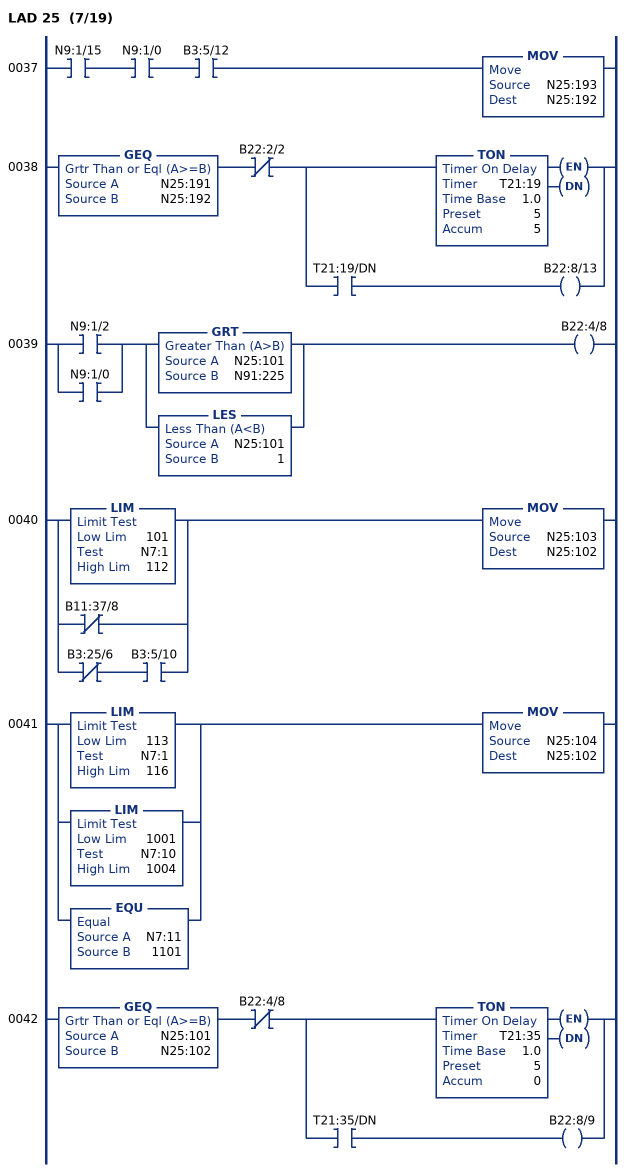
% Rung: 37 %
SOR XIC N9:1/15 XIC N9:1/0 XIC B3:5/12 MOV N25:193 N25:192 EOR
% Rung: 38 %
SOR GEQ N25:191 N25:192 XIO B22:2/2 BST TON T21:19 1.0 5 5 NXB XIC T21:19/DN OTE B22:8/13 BND EOR
% Rung: 39 %
SOR BST XIC N9:1/2 NXB XIC N9:1/0 BND BST GRT N25:101 N91:225 NXB LES N25:101 1 BND OTE B22:4/8 EOR
% Rung: 40 %
SOR BST LIM 101 N7:1 112 NXB XIO B11:37/8 NXB XIO B3:25/6 XIC B3:5/10 BND MOV N25:103 N25:102 EOR
% Rung: 41 %
SOR BST LIM 113 N7:1 116 NXB LIM 1001 N7:10 1004 NXB EQU N7:11 1101 BND MOV N25:104 N25:102 EOR
% Rung: 42 %
SOR GEQ N25:101 N25:102 XIO B22:4/8 BST TON T21:35 1.0 5 0 NXB XIC T21:35/DN OTE B22:8/9 BND EOR

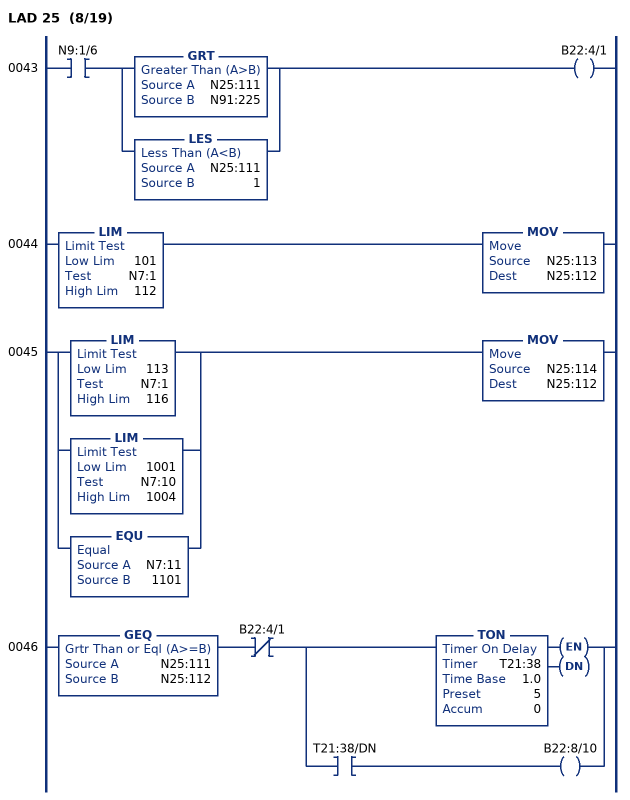
% Rung: 43 %
SOR XIC N9:1/6 BST GRT N25:111 N91:225 NXB LES N25:111 1 BND OTE B22:4/1 EOR
% Rung: 44 %
SOR LIM 101 N7:1 112 MOV N25:113 N25:112 EOR
% Rung: 45 %
SOR BST LIM 113 N7:1 116 NXB LIM 1001 N7:10 1004 NXB EQU N7:11 1101 BND MOV N25:114 N25:112 EOR
% Rung: 46 %
SOR GEQ N25:111 N25:112 XIO B22:4/1 BST TON T21:38 1.0 5 0 NXB XIC T21:38/DN OTE B22:8/10 BND EOR

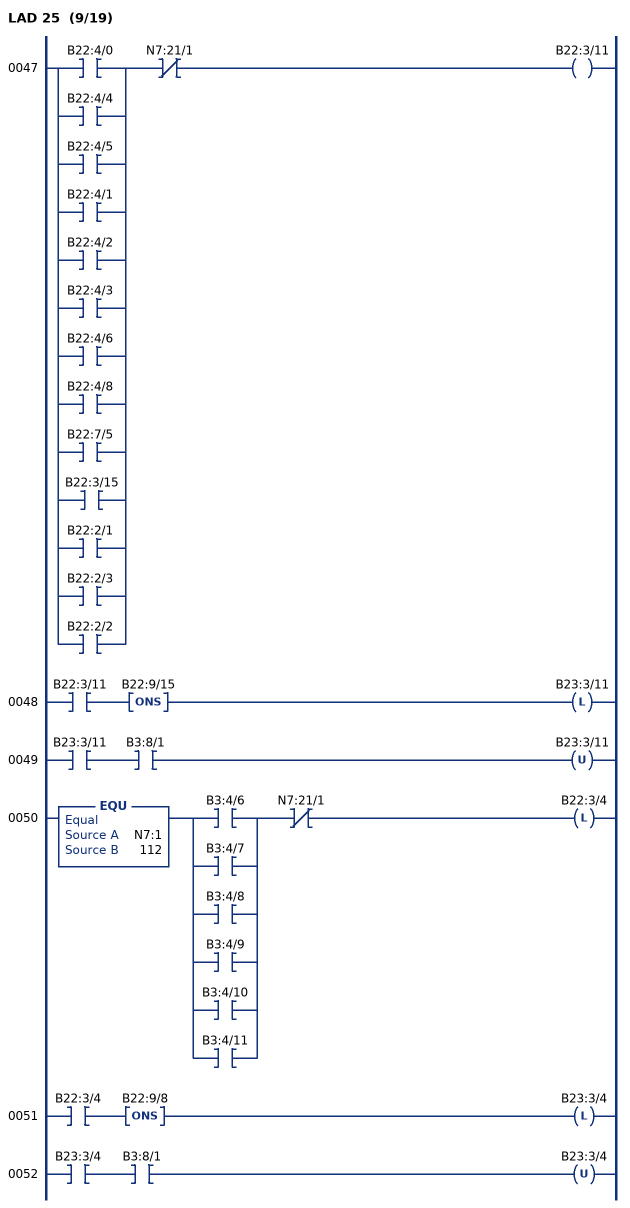
% Rung: 47 %
SOR BST XIC B22:4/0 NXB XIC B22:4/4 NXB XIC B22:4/5 NXB XIC B22:4/1 NXB XIC B22:4/2 NXB XIC B22:4/3 NXB XIC B22:4/6 NXB XIC B22:4/8 NXB XIC B22:7/5 NXB XIC B22:3/15 NXB XIC B22:2/1 NXB XIC B22:2/3 NXB XIC B22:2/2 BND XIO N7:21/1 OTE B22:3/11 EOR
% Rung: 48 %
SOR XIC B22:3/11 OSR B22:9/15 OTL B23:3/11 EOR
% Rung: 49 %
SOR XIC B23:3/11 XIC B3:8/1 OTU B23:3/11 EOR
% Rung: 50 %
SOR EQU N7:1 112 BST XIC B3:4/6 NXB XIC B3:4/7 NXB XIC B3:4/8 NXB XIC B3:4/9 NXB XIC B3:4/10 NXB XIC B3:4/11 BND XIO N7:21/1 OTL B22:3/4 EOR
% Rung: 51 %
SOR XIC B22:3/4 OSR B22:9/8 OTL B23:3/4 EOR
% Rung: 52 %
SOR XIC B23:3/4 XIC B3:8/1 OTU B23:3/4 EOR

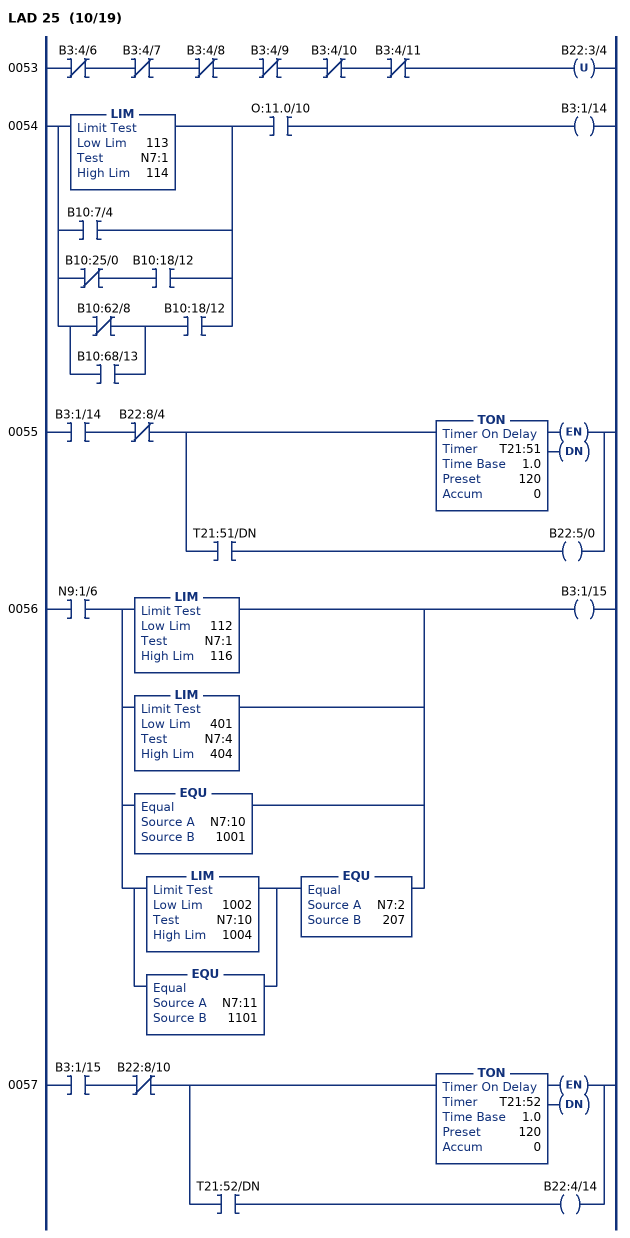
% Rung: 53 %
SOR XIO B3:4/6 XIO B3:4/7 XIO B3:4/8 XIO B3:4/9 XIO B3:4/10 XIO B3:4/11 OTU B22:3/4 EOR
% Rung: 54 %
SOR BST LIM 113 N7:1 114 NXB XIC B10:7/4 NXB XIO B10:25/0 XIC B10:18/12 NXB BST XIO B10:62/8 NXB XIC B10:68/13 BND XIC B10:18/12 BND XIC O:11.0/10 OTE B3:1/14 EOR
% Rung: 55 %
SOR XIC B3:1/14 XIO B22:8/4 BST TON T21:51 1.0 120 0 NXB XIC T21:51/DN OTE B22:5/0 BND EOR
% Rung: 56 %
SOR XIC N9:1/6 BST LIM 112 N7:1 116 NXB LIM 401 N7:4 404 NXB EQU N7:10 1001 NXB BST LIM 1002 N7:10 1004 NXB EQU N7:11 1101 BND EQU N7:2 207 BND OTE B3:1/15 EOR
% Rung: 57 %
SOR XIC B3:1/15 XIO B22:8/10 BST TON T21:52 1.0 120 0 NXB XIC T21:52/DN OTE B22:4/14 BND EOR

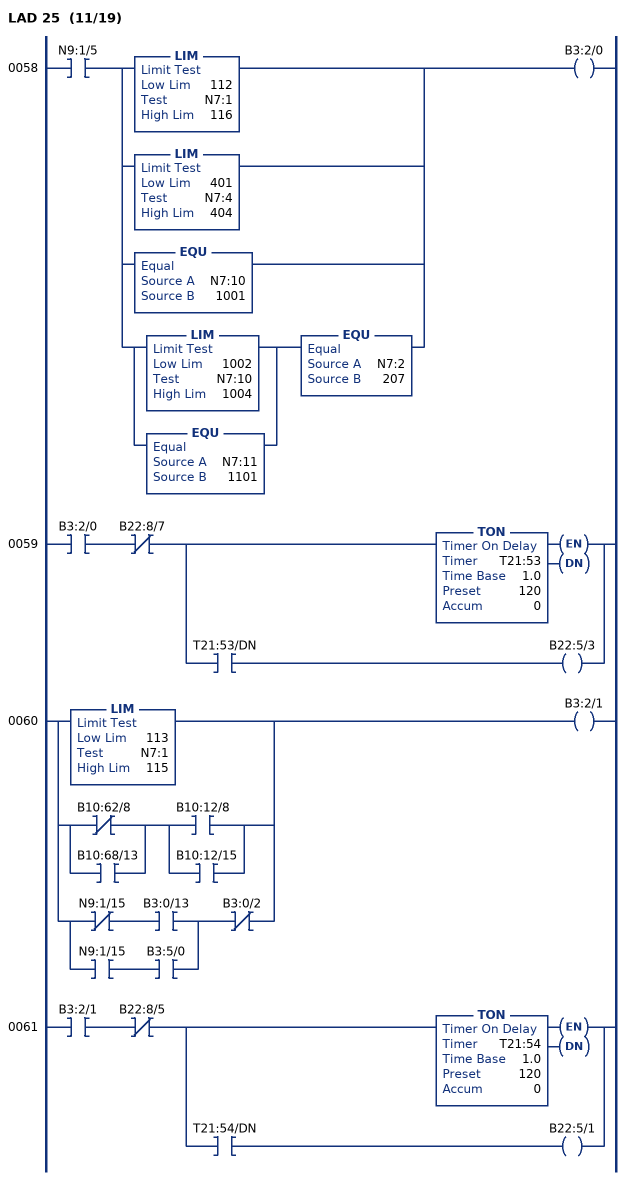
% Rung: 58 %
SOR XIC N9:1/5 BST LIM 112 N7:1 116 NXB LIM 401 N7:4 404 NXB EQU N7:10 1001 NXB BST LIM 1002 N7:10 1004 NXB EQU N7:11 1101 BND EQU N7:2 207 BND OTE B3:2/0 EOR
% Rung: 59 %
SOR XIC B3:2/0 XIO B22:8/7 BST TON T21:53 1.0 120 0 NXB XIC T21:53/DN OTE B22:5/3 BND EOR
% Rung: 60 %
SOR BST LIM 113 N7:1 115 NXB BST XIO B10:62/8 NXB XIC B10:68/13 BND BST XIC B10:12/8 NXB XIC B10:12/15 BND NXB BST XIO N9:1/15 XIC B3:0/13 NXB XIC N9:1/15 XIC B3:5/0 BND XIO B3:0/2 BND OTE B3:2/1 EOR
% Rung: 61 %
SOR XIC B3:2/1 XIO B22:8/5 BST TON T21:54 1.0 120 0 NXB XIC T21:54/DN OTE B22:5/1 BND EOR

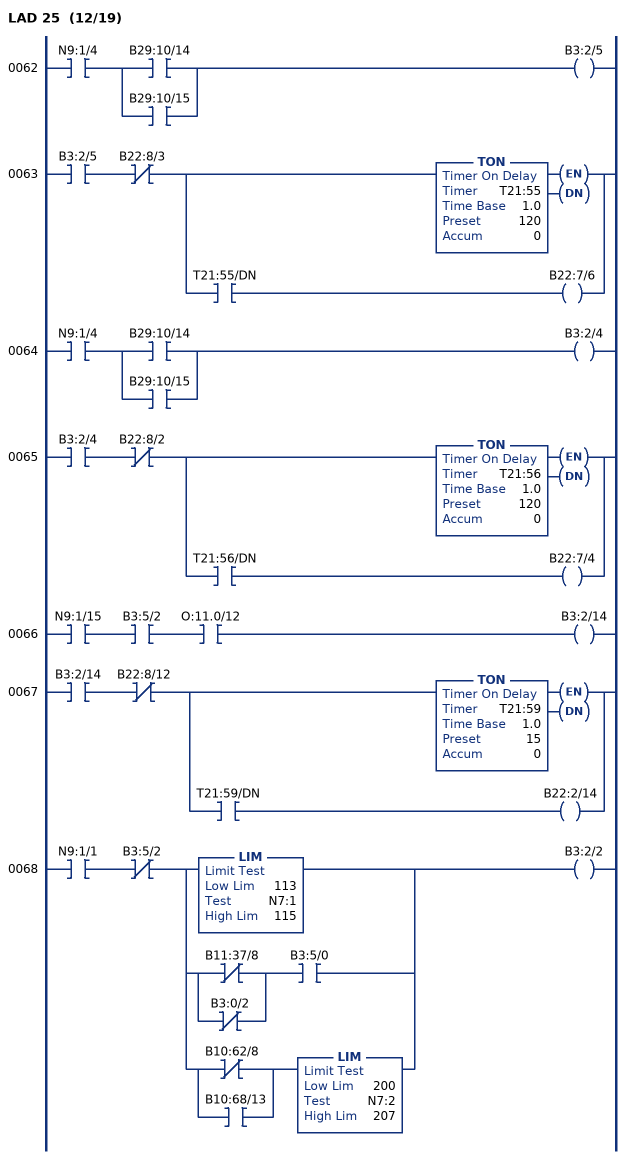
% Rung: 62 %
SOR XIC N9:1/4 BST XIC B29:10/14 NXB XIC B29:10/15 BND OTE B3:2/5 EOR
% Rung: 63 %
SOR XIC B3:2/5 XIO B22:8/3 BST TON T21:55 1.0 120 0 NXB XIC T21:55/DN OTE B22:7/6 BND EOR
% Rung: 64 %
SOR XIC N9:1/4 BST XIC B29:10/14 NXB XIC B29:10/15 BND OTE B3:2/4 EOR
% Rung: 65 %
SOR XIC B3:2/4 XIO B22:8/2 BST TON T21:56 1.0 120 0 NXB XIC T21:56/DN OTE B22:7/4 BND EOR
% Rung: 66 %
SOR XIC N9:1/15 XIC B3:5/2 XIC O:11.0/12 OTE B3:2/14 EOR
% Rung: 67 %
SOR XIC B3:2/14 XIO B22:8/12 BST TON T21:59 1.0 15 0 NXB XIC T21:59/DN OTE B22:2/14 BND EOR
% Rung: 68 %
SOR XIC N9:1/1 XIO B3:5/2 BST LIM 113 N7:1 115 NXB BST XIO B11:37/8 NXB XIO B3:0/2 BND XIC B3:5/0 NXB BST XIO B10:62/8 NXB XIC B10:68/13 BND LIM 200 N7:2 207 BND OTE B3:2/2 EOR

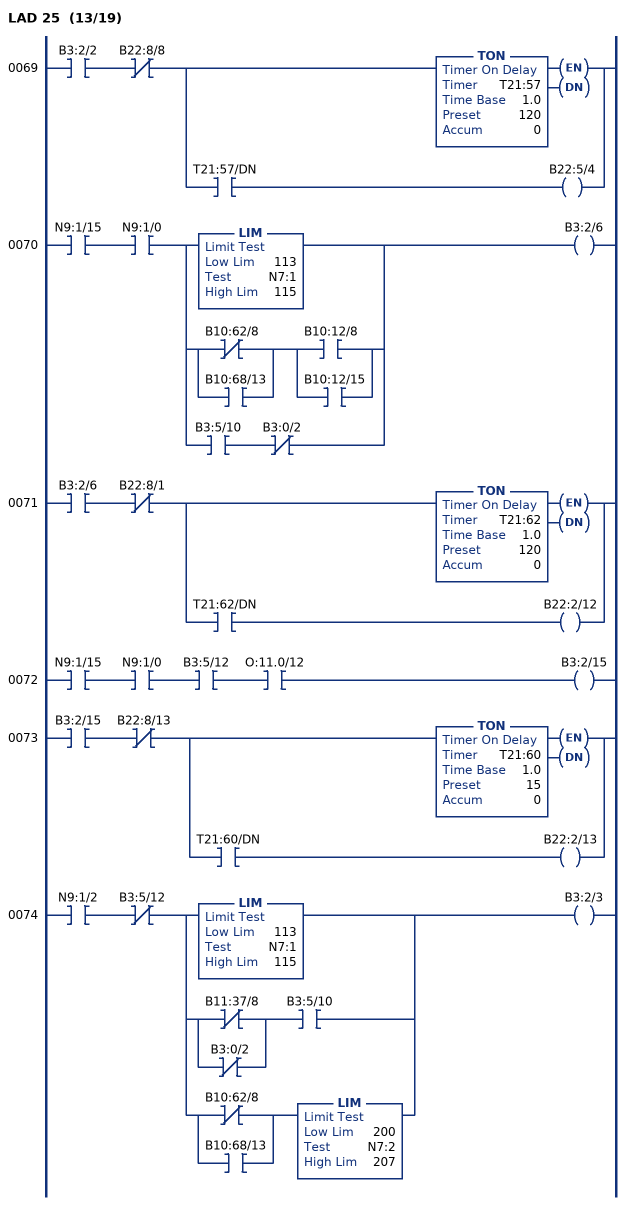
% Rung: 69 %
SOR XIC B3:2/2 XIO B22:8/8 BST TON T21:57 1.0 120 0 NXB XIC T21:57/DN OTE B22:5/4 BND EOR
% Rung: 70 %
SOR XIC N9:1/15 XIC N9:1/0 BST LIM 113 N7:1 115 NXB BST XIO B10:62/8 NXB XIC B10:68/13 BND BST XIC B10:12/8 NXB XIC B10:12/15 BND NXB XIC B3:5/10 XIO B3:0/2 BND OTE B3:2/6 EOR
% Rung: 71 %
SOR XIC B3:2/6 XIO B22:8/1 BST TON T21:62 1.0 120 0 NXB XIC T21:62/DN OTE B22:2/12 BND EOR
% Rung: 72 %
SOR XIC N9:1/15 XIC N9:1/0 XIC B3:5/12 XIC O:11.0/12 OTE B3:2/15 EOR
% Rung: 73 %
SOR XIC B3:2/15 XIO B22:8/13 BST TON T21:60 1.0 15 0 NXB XIC T21:60/DN OTE B22:2/13 BND EOR
% Rung: 74 %
SOR XIC N9:1/2 XIO B3:5/12 BST LIM 113 N7:1 115 NXB BST XIO B11:37/8 NXB XIO B3:0/2 BND XIC B3:5/10 NXB BST XIO B10:62/8 NXB XIC B10:68/13 BND LIM 200 N7:2 207 BND OTE B3:2/3 EOR

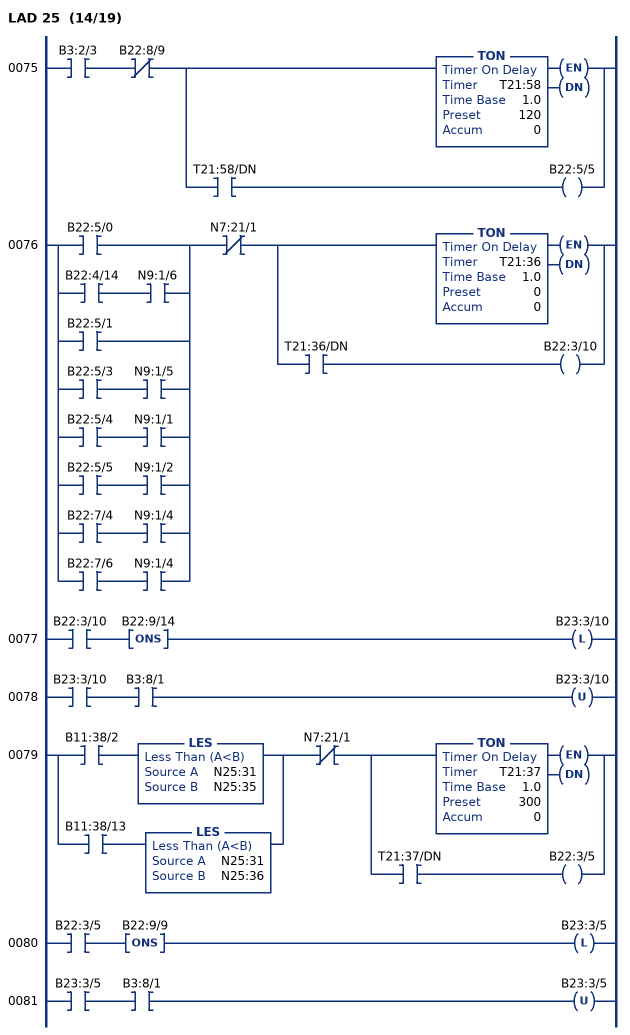
% Rung: 75 %
SOR XIC B3:2/3 XIO B22:8/9 BST TON T21:58 1.0 120 0 NXB XIC T21:58/DN OTE B22:5/5 BND EOR
% Rung: 76 %
SOR BST XIC B22:5/0 NXB XIC B22:4/14 XIC N9:1/6 NXB XIC B22:5/1 NXB XIC B22:5/3 XIC N9:1/5 NXB XIC B22:5/4 XIC N9:1/1 NXB XIC B22:5/5 XIC N9:1/2 NXB XIC B22:7/4 XIC N9:1/4 NXB XIC B22:7/6 XIC N9:1/4 BND XIO N7:21/1 BST TON T21:36 1.0 0 0 NXB XIC T21:36/DN OTE B22:3/10 BND EOR
% Rung: 77 %
SOR XIC B22:3/10 OSR B22:9/14 OTL B23:3/10 EOR
% Rung: 78 %
SOR XIC B23:3/10 XIC B3:8/1 OTU B23:3/10 EOR
% Rung: 79 %
SOR BST XIC B11:38/2 LES N25:31 N25:35 NXB XIC B11:38/13 LES N25:31 N25:36 BND XIO N7:21/1 BST TON T21:37 1.0 300 0 NXB XIC T21:37/DN OTE B22:3/5 BND EOR
% Rung: 80 %
SOR XIC B22:3/5 OSR B22:9/9 OTL B23:3/5 EOR
% Rung: 81 %
SOR XIC B23:3/5 XIC B3:8/1 OTU B23:3/5 EOR

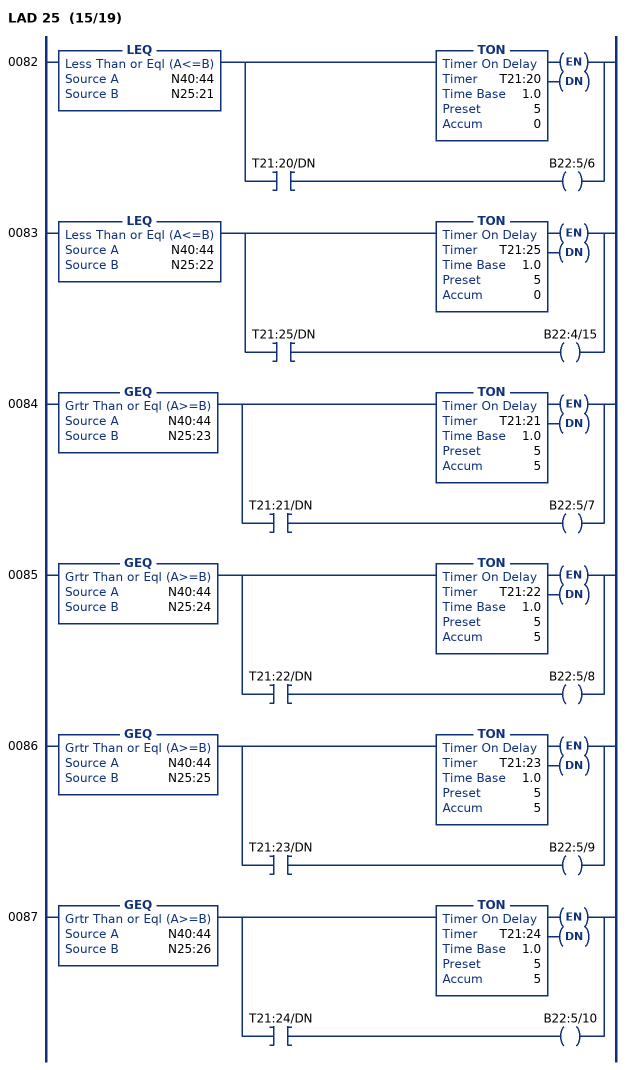
% Rung: 82 %
SOR LEQ N40:44 N25:21 BST TON T21:20 1.0 5 0 NXB XIC T21:20/DN OTE B22:5/6 BND EOR
% Rung: 83 %
SOR LEQ N40:44 N25:22 BST TON T21:25 1.0 5 0 NXB XIC T21:25/DN OTE B22:4/15 BND EOR
% Rung: 84 %
SOR GEQ N40:44 N25:23 BST TON T21:21 1.0 5 5 NXB XIC T21:21/DN OTE B22:5/7 BND EOR
% Rung: 85 %
SOR GEQ N40:44 N25:24 BST TON T21:22 1.0 5 5 NXB XIC T21:22/DN OTE B22:5/8 BND EOR
% Rung: 86 %
SOR GEQ N40:44 N25:25 BST TON T21:23 1.0 5 5 NXB XIC T21:23/DN OTE B22:5/9 BND EOR
% Rung: 87 %
SOR GEQ N40:44 N25:26 BST TON T21:24 1.0 5 5 NXB XIC T21:24/DN OTE B22:5/10 BND EOR

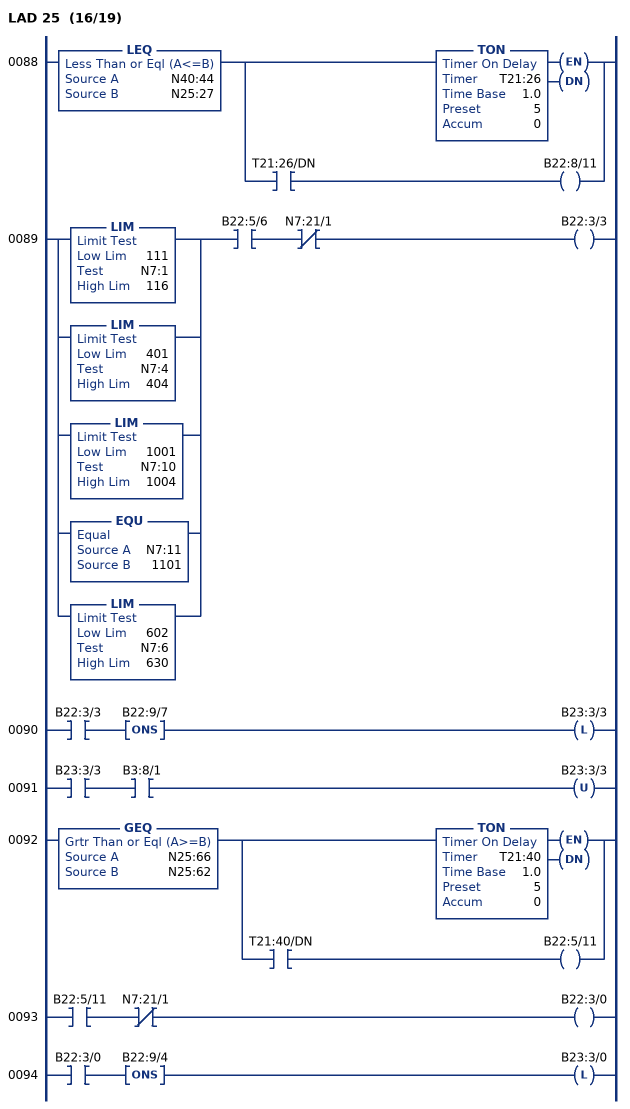
% Rung: 88 %
SOR LEQ N40:44 N25:27 BST TON T21:26 1.0 5 0 NXB XIC T21:26/DN OTE B22:8/11 BND EOR
% Rung: 89 %
SOR BST LIM 111 N7:1 116 NXB LIM 401 N7:4 404 NXB LIM 1001 N7:10 1004 NXB EQU N7:11 1101 NXB LIM 602 N7:6 630 BND XIC B22:5/6 XIO N7:21/1 OTE B22:3/3 EOR
% Rung: 90 %
SOR XIC B22:3/3 OSR B22:9/7 OTL B23:3/3 EOR
% Rung: 91 %
SOR XIC B23:3/3 XIC B3:8/1 OTU B23:3/3 EOR
% Rung: 92 %
SOR GEQ N25:66 N25:62 BST TON T21:40 1.0 5 0 NXB XIC T21:40/DN OTE B22:5/11 BND EOR
% Rung: 93 %
SOR XIC B22:5/11 XIO N7:21/1 OTE B22:3/0 EOR
% Rung: 94 %
SOR XIC B22:3/0 OSR B22:9/4 OTL B23:3/0 EOR

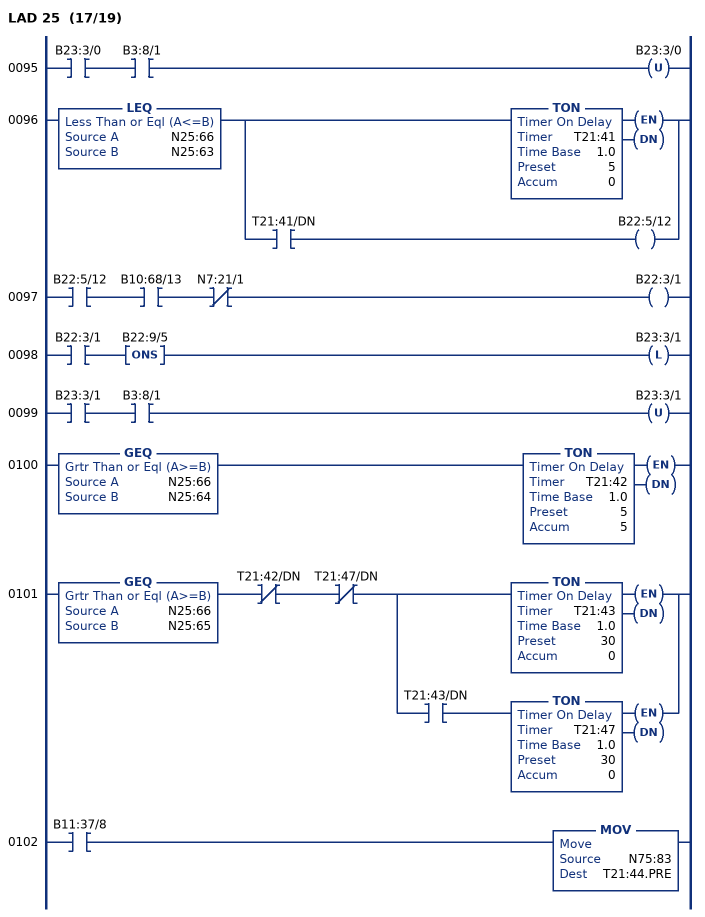
% Rung: 95 %
SOR XIC B23:3/0 XIC B3:8/1 OTU B23:3/0 EOR
% Rung: 96 %
SOR LEQ N25:66 N25:63 BST TON T21:41 1.0 5 0 NXB XIC T21:41/DN OTE B22:5/12 BND EOR
% Rung: 97 %
SOR XIC B22:5/12 XIC B10:68/13 XIO N7:21/1 OTE B22:3/1 EOR
% Rung: 98 %
SOR XIC B22:3/1 OSR B22:9/5 OTL B23:3/1 EOR
% Rung: 99 %
SOR XIC B23:3/1 XIC B3:8/1 OTU B23:3/1 EOR
% Rung: 100 %
SOR GEQ N25:66 N25:64 TON T21:42 1.0 5 5 EOR
% Rung: 101 %
SOR GEQ N25:66 N25:65 XIO T21:42/DN XIO T21:47/DN BST TON T21:43 1.0 30 0 NXB XIC T21:43/DN TON T21:47 1.0 30 0 BND EOR
% Rung: 102 %
SOR XIC B11:37/8 MOV N75:83 T21:44.PRE EOR

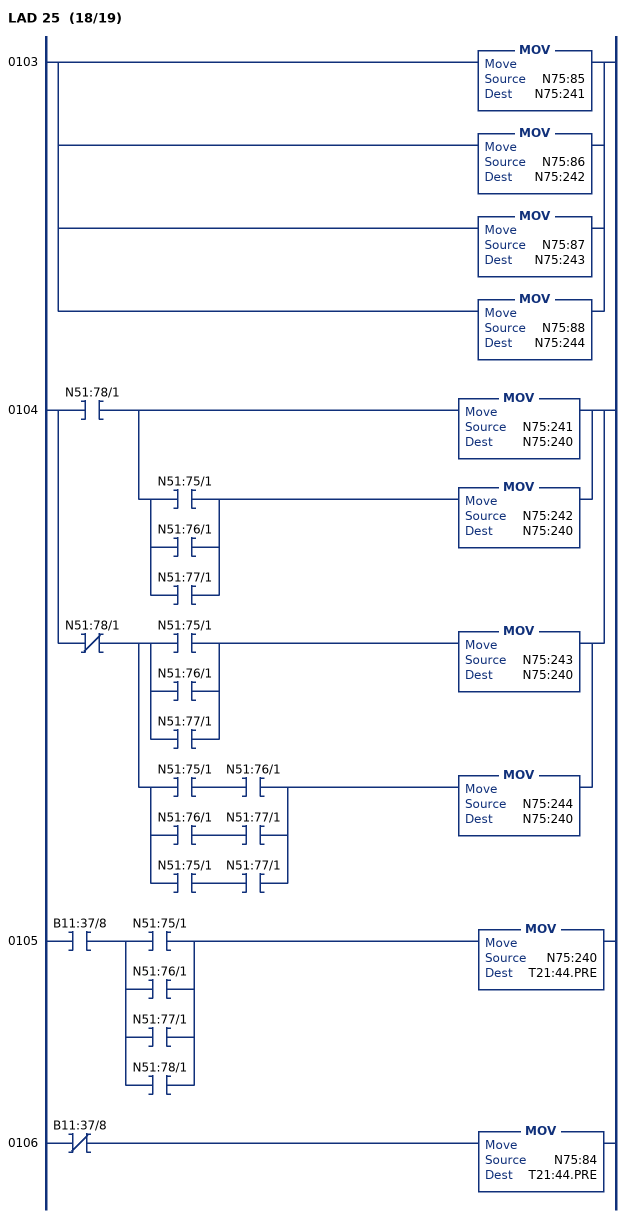
% Rung: 103 %
SOR BST MOV N75:85 N75:241 NXB BST MOV N75:86 N75:242 NXB BST MOV N75:87 N75:243 NXB MOV N75:88 N75:244 BND BND BND EOR
% Rung: 104 %
SOR BST XIC N51:78/1 BST MOV N75:241 N75:240 NXB BST XIC N51:75/1 NXB BST XIC N51:76/1 NXB XIC N51:77/1 BND BND MOV N75:242 N75:240 BND NXB XIO N51:78/1 BST BST XIC N51:75/1 NXB BST XIC N51:76/1 NXB XIC N51:77/1 BND BND MOV N75:243 N75:240 NXB BST XIC N51:75/1 XIC N51:76/1 NXB BST XIC N51:76/1 XIC N51:77/1 NXB XIC N51:75/1 XIC N51:77/1 BND BND MOV N75:244 N75:240 BND BND EOR
% Rung: 105 %
SOR XIC B11:37/8 BST XIC N51:75/1 NXB BST XIC N51:76/1 NXB BST XIC N51:77/1 NXB XIC N51:78/1 BND BND BND MOV N75:240 T21:44.PRE EOR
% Rung: 106 %
SOR XIO B11:37/8 MOV N75:84 T21:44.PRE EOR

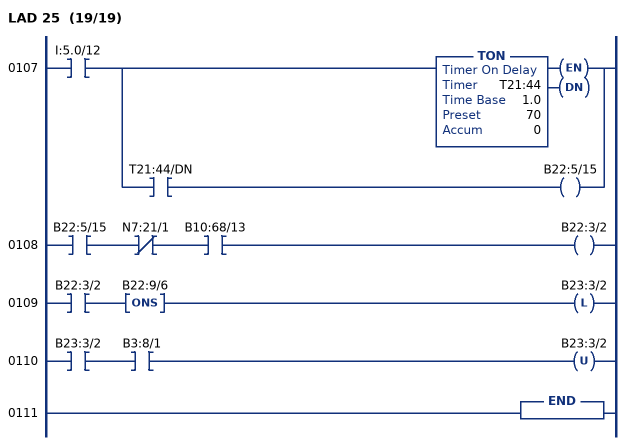
% Rung: 107 %
SOR XIC I:5.0/12 BST TON T21:44 1.0 70 0 NXB XIC T21:44/DN OTE B22:5/15 BND EOR
% Rung: 108 %
SOR XIC B22:5/15 XIO N7:21/1 XIC B10:68/13 OTE B22:3/2 EOR
% Rung: 109 %
SOR XIC B22:3/2 OSR B22:9/6 OTL B23:3/2 EOR
% Rung: 110 %
SOR XIC B23:3/2 XIC B3:8/1 OTU B23:3/2 EOR
% Rung: 111 %
SOR END EOR

LADDER 26
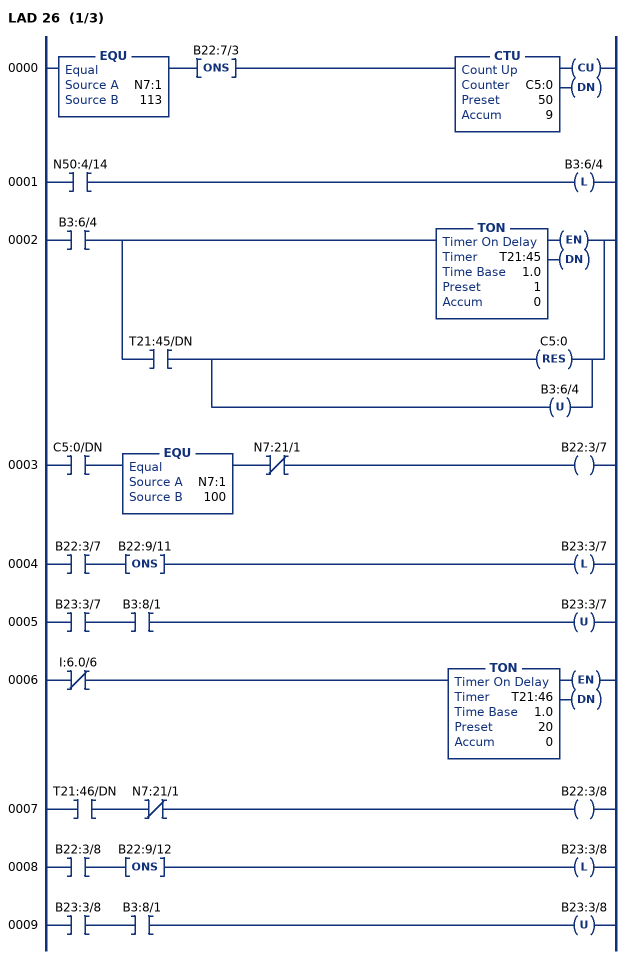
% Rung: 0 %
SOR EQU N7:1 113 OSR B22:7/3 CTU C5:0 50 9 EOR
% Rung: 1 %
SOR XIC N50:4/14 OTL B3:6/4 EOR
% Rung: 2 %
SOR XIC B3:6/4 BST TON T21:45 1.0 1 0 NXB XIC T21:45/DN BST RES C5:0 NXB OTU B3:6/4 BND BND EOR
% Rung: 3 %
SOR XIC C5:0/DN EQU N7:1 100 XIO N7:21/1 OTE B22:3/7 EOR
% Rung: 4 %
SOR XIC B22:3/7 OSR B22:9/11 OTL B23:3/7 EOR
% Rung: 5 %
SOR XIC B23:3/7 XIC B3:8/1 OTU B23:3/7 EOR
% Rung: 6 %
SOR XIO I:6.0/6 TON T21:46 1.0 20 0 EOR
% Rung: 7 %
SOR XIC T21:46/DN XIO N7:21/1 OTE B22:3/8 EOR
% Rung: 8 %
SOR XIC B22:3/8 OSR B22:9/12 OTL B23:3/8 EOR
% Rung: 9 %
SOR XIC B23:3/8 XIC B3:8/1 OTU B23:3/8 EOR

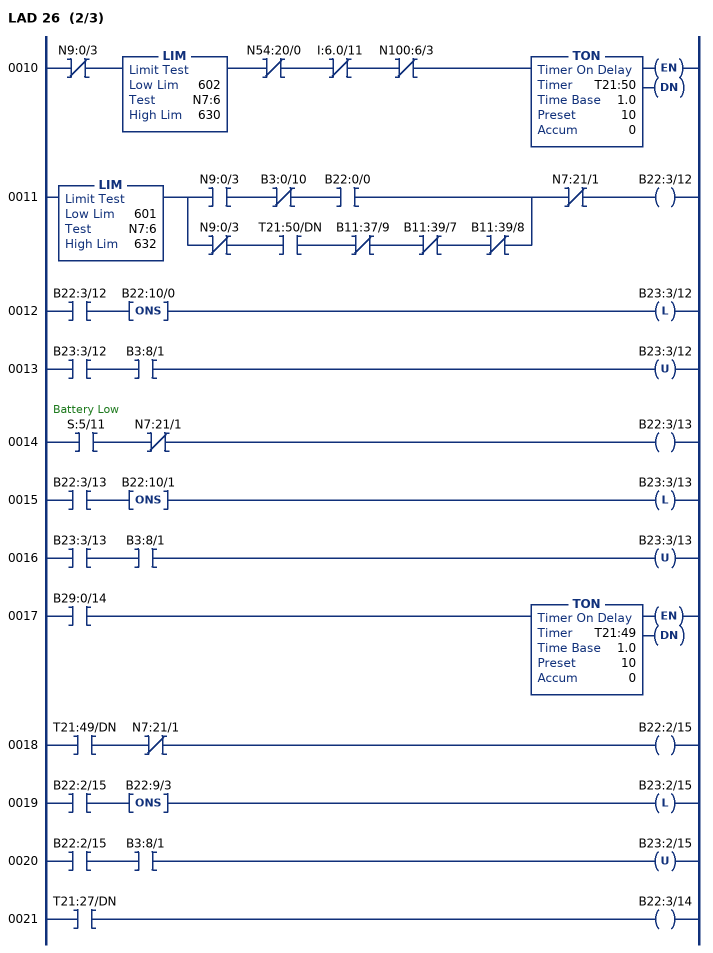
% Rung: 10 %
SOR XIO N9:0/3 LIM 602 N7:6 630 XIO N54:20/0 XIO I:6.0/11 XIO N100:6/3 TON T21:50 1.0 10 0 EOR
% Rung: 11 %
SOR LIM 601 N7:6 632 BST XIC N9:0/3 XIO B3:0/10 XIC B22:0/0 NXB XIO N9:0/3 XIC T21:50/DN XIO B11:37/9 XIO B11:39/7 XIO B11:39/8 BND XIO N7:21/1 OTE B22:3/12 EOR
% Rung: 12 %
SOR XIC B22:3/12 OSR B22:10/0 OTL B23:3/12 EOR
% Rung: 13 %
SOR XIC B23:3/12 XIC B3:8/1 OTU B23:3/12 EOR
% Rung: 14 %
SOR XIC S:5/11 XIO N7:21/1 OTE B22:3/13 EOR
%   S:5/11  "Battery Low" %
% Rung: 15 %
SOR XIC B22:3/13 OSR B22:10/1 OTL B23:3/13 EOR
% Rung: 16 %
SOR XIC B23:3/13 XIC B3:8/1 OTU B23:3/13 EOR
% Rung: 17 %
SOR XIC B29:0/14 TON T21:49 1.0 10 0 EOR
% Rung: 18 %
SOR XIC T21:49/DN XIO N7:21/1 OTE B22:2/15 EOR
% Rung: 19 %
SOR XIC B22:2/15 OSR B22:9/3 OTL B23:2/15 EOR
% Rung: 20 %
SOR XIC B22:2/15 XIC B3:8/1 OTU B23:2/15 EOR
% Rung: 21 %
SOR XIC T21:27/DN OTE B22:3/14 EOR

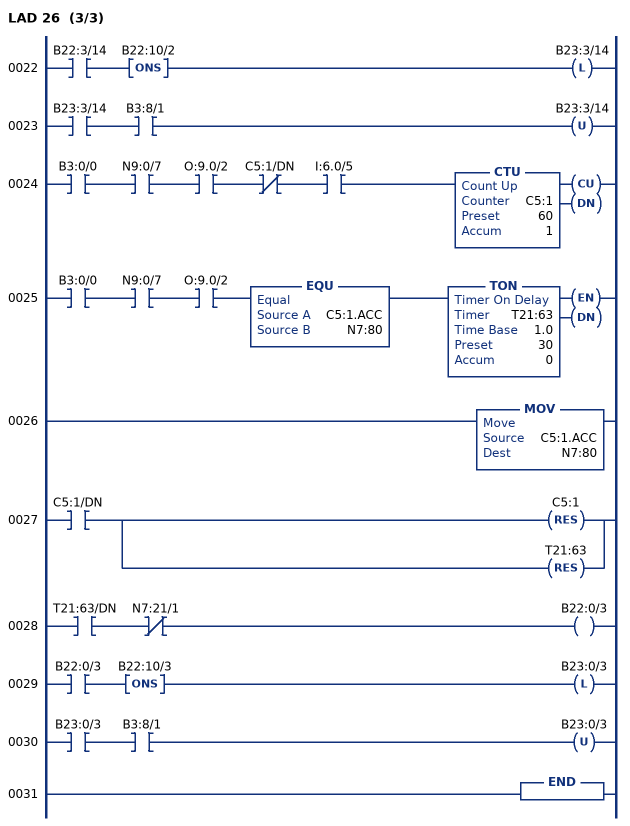
% Rung: 22 %
SOR XIC B22:3/14 OSR B22:10/2 OTL B23:3/14 EOR
% Rung: 23 %
SOR XIC B23:3/14 XIC B3:8/1 OTU B23:3/14 EOR
% Rung: 24 %
SOR XIC B3:0/0 XIC N9:0/7 XIC O:9.0/2 XIO C5:1/DN XIC I:6.0/5 CTU C5:1 60 1 EOR
% Rung: 25 %
SOR XIC B3:0/0 XIC N9:0/7 XIC O:9.0/2 EQU C5:1.ACC N7:80 TON T21:63 1.0 30 0 EOR
% Rung: 26 %
SOR MOV C5:1.ACC N7:80 EOR
% Rung: 27 %
SOR XIC C5:1/DN BST RES C5:1 NXB RES T21:63 BND EOR
% Rung: 28 %
SOR XIC T21:63/DN XIO N7:21/1 OTE B22:0/3 EOR
% Rung: 29 %
SOR XIC B22:0/3 OSR B22:10/3 OTL B23:0/3 EOR
% Rung: 30 %
SOR XIC B23:0/3 XIC B3:8/1 OTU B23:0/3 EOR
% Rung: 31 %
SOR END EOR

LADDER 27
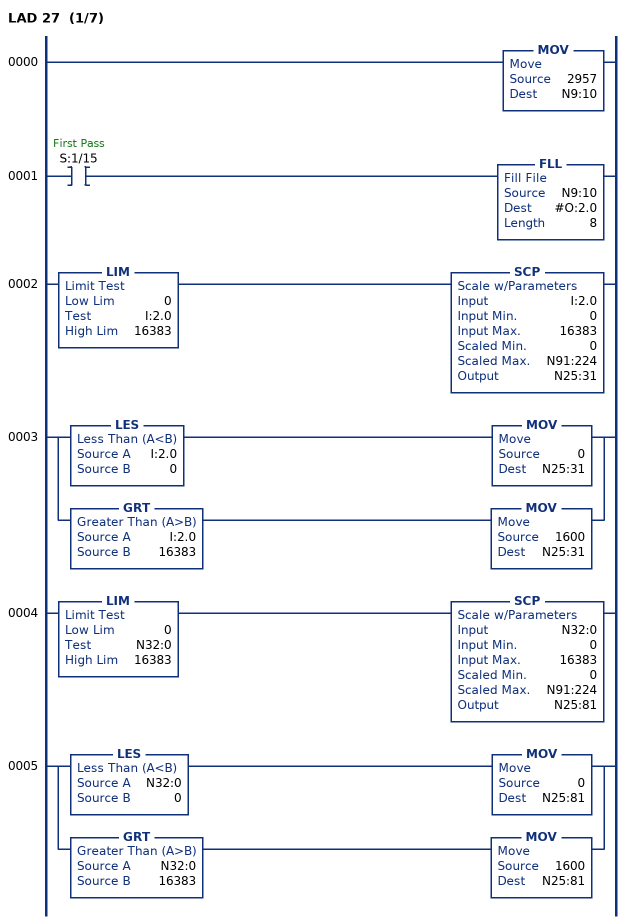
% Rung: 0 %
SOR MOV 2957 N9:10 EOR
% Rung: 1 %
SOR XIC S:1/15 FLL N9:10 #O:2.0 8 EOR
%   S:1/15  "First Pass" %
% Rung: 2 %
SOR LIM 0 I:2.0 16383 SCP I:2.0 0 16383 0 N91:224 N25:31 EOR
% Rung: 3 %
SOR BST LES I:2.0 0 MOV 0 N25:31 NXB GRT I:2.0 16383 MOV 1600 N25:31 BND EOR
% Rung: 4 %
SOR LIM 0 N32:0 16383 SCP N32:0 0 16383 0 N91:224 N25:81 EOR
% Rung: 5 %
SOR BST LES N32:0 0 MOV 0 N25:81 NXB GRT N32:0 16383 MOV 1600 N25:81 BND EOR

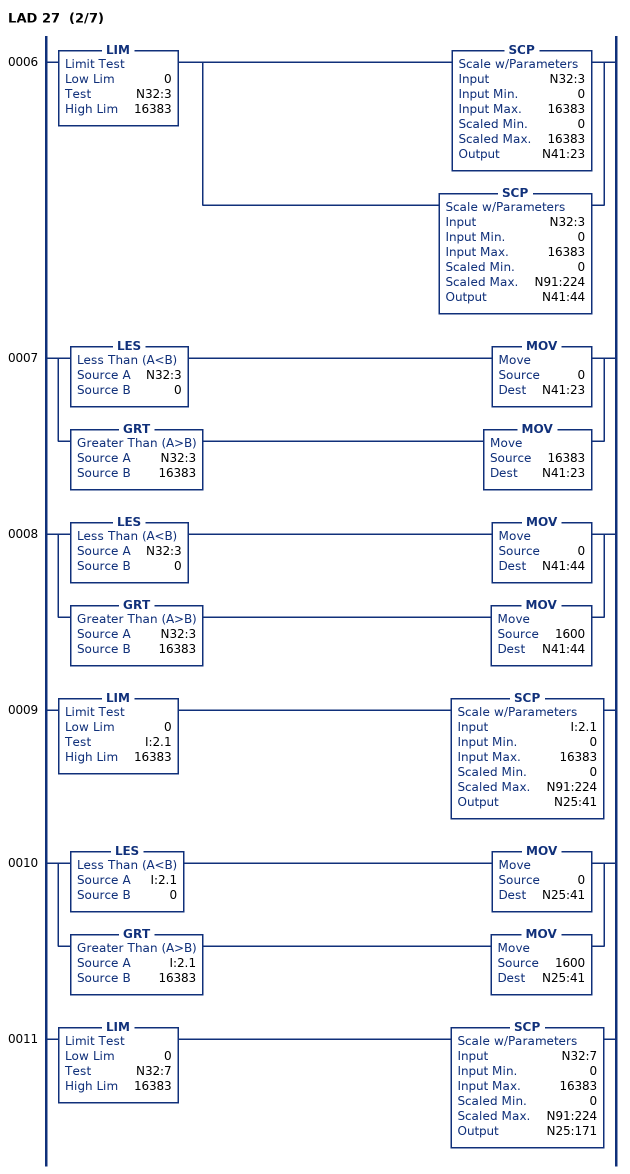
% Rung: 6 %
SOR LIM 0 N32:3 16383 BST SCP N32:3 0 16383 0 16383 N41:23 NXB SCP N32:3 0 16383 0 N91:224 N41:44 BND EOR
% Rung: 7 %
SOR BST LES N32:3 0 MOV 0 N41:23 NXB GRT N32:3 16383 MOV 16383 N41:23 BND EOR
% Rung: 8 %
SOR BST LES N32:3 0 MOV 0 N41:44 NXB GRT N32:3 16383 MOV 1600 N41:44 BND EOR
% Rung: 9 %
SOR LIM 0 I:2.1 16383 SCP I:2.1 0 16383 0 N91:224 N25:41 EOR
% Rung: 10 %
SOR BST LES I:2.1 0 MOV 0 N25:41 NXB GRT I:2.1 16383 MOV 1600 N25:41 BND EOR
% Rung: 11 %
SOR LIM 0 N32:7 16383 SCP N32:7 0 16383 0 N91:224 N25:171 EOR

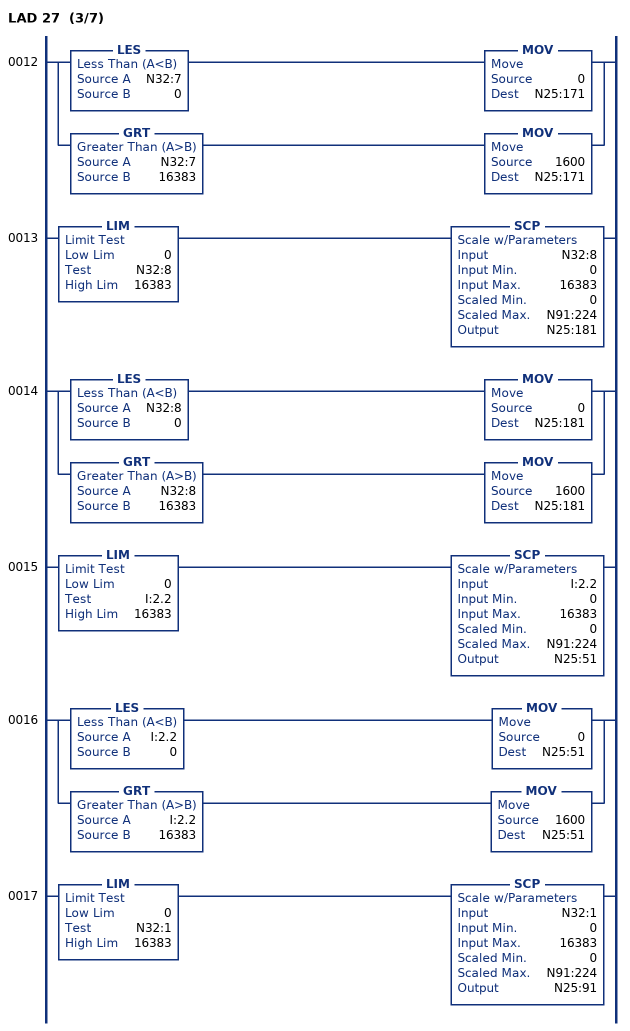
% Rung: 12 %
SOR BST LES N32:7 0 MOV 0 N25:171 NXB GRT N32:7 16383 MOV 1600 N25:171 BND EOR
% Rung: 13 %
SOR LIM 0 N32:8 16383 SCP N32:8 0 16383 0 N91:224 N25:181 EOR
% Rung: 14 %
SOR BST LES N32:8 0 MOV 0 N25:181 NXB GRT N32:8 16383 MOV 1600 N25:181 BND EOR
% Rung: 15 %
SOR LIM 0 I:2.2 16383 SCP I:2.2 0 16383 0 N91:224 N25:51 EOR
% Rung: 16 %
SOR BST LES I:2.2 0 MOV 0 N25:51 NXB GRT I:2.2 16383 MOV 1600 N25:51 BND EOR
% Rung: 17 %
SOR LIM 0 N32:1 16383 SCP N32:1 0 16383 0 N91:224 N25:91 EOR

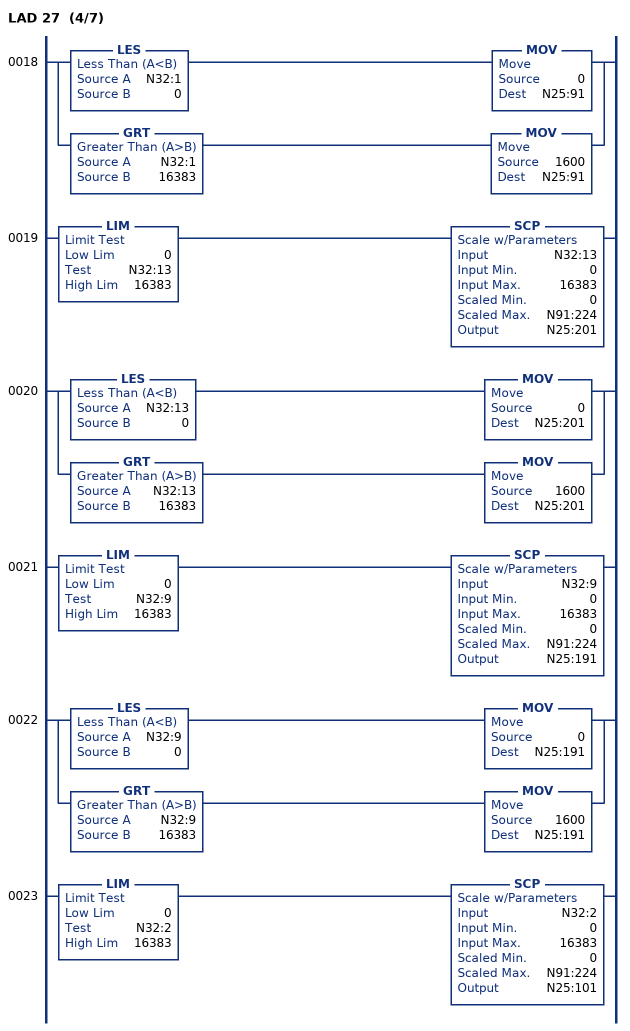
% Rung: 18 %
SOR BST LES N32:1 0 MOV 0 N25:91 NXB GRT N32:1 16383 MOV 1600 N25:91 BND EOR
% Rung: 19 %
SOR LIM 0 N32:13 16383 SCP N32:13 0 16383 0 N91:224 N25:201 EOR
% Rung: 20 %
SOR BST LES N32:13 0 MOV 0 N25:201 NXB GRT N32:13 16383 MOV 1600 N25:201 BND EOR
% Rung: 21 %
SOR LIM 0 N32:9 16383 SCP N32:9 0 16383 0 N91:224 N25:191 EOR
% Rung: 22 %
SOR BST LES N32:9 0 MOV 0 N25:191 NXB GRT N32:9 16383 MOV 1600 N25:191 BND EOR
% Rung: 23 %
SOR LIM 0 N32:2 16383 SCP N32:2 0 16383 0 N91:224 N25:101 EOR

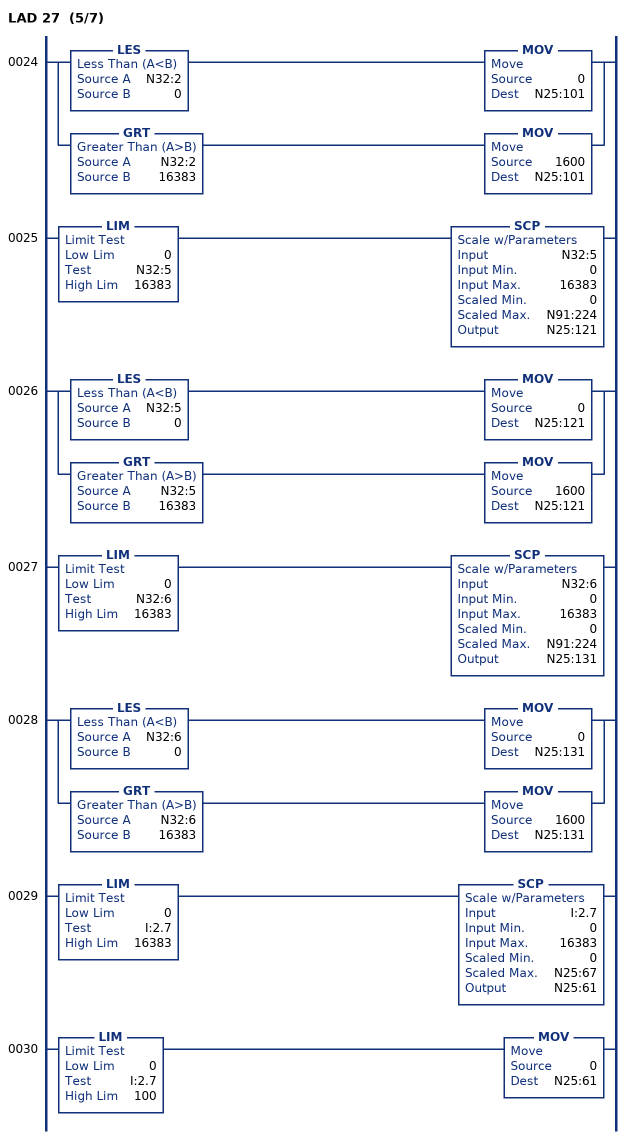
% Rung: 24 %
SOR BST LES N32:2 0 MOV 0 N25:101 NXB GRT N32:2 16383 MOV 1600 N25:101 BND EOR
% Rung: 25 %
SOR LIM 0 N32:5 16383 SCP N32:5 0 16383 0 N91:224 N25:121 EOR
% Rung: 26 %
SOR BST LES N32:5 0 MOV 0 N25:121 NXB GRT N32:5 16383 MOV 1600 N25:121 BND EOR
% Rung: 27 %
SOR LIM 0 N32:6 16383 SCP N32:6 0 16383 0 N91:224 N25:131 EOR
% Rung: 28 %
SOR BST LES N32:6 0 MOV 0 N25:131 NXB GRT N32:6 16383 MOV 1600 N25:131 BND EOR
% Rung: 29 %
SOR LIM 0 I:2.7 16383 SCP I:2.7 0 16383 0 N25:67 N25:61 EOR
% Rung: 30 %
SOR LIM 0 I:2.7 100 MOV 0 N25:61 EOR

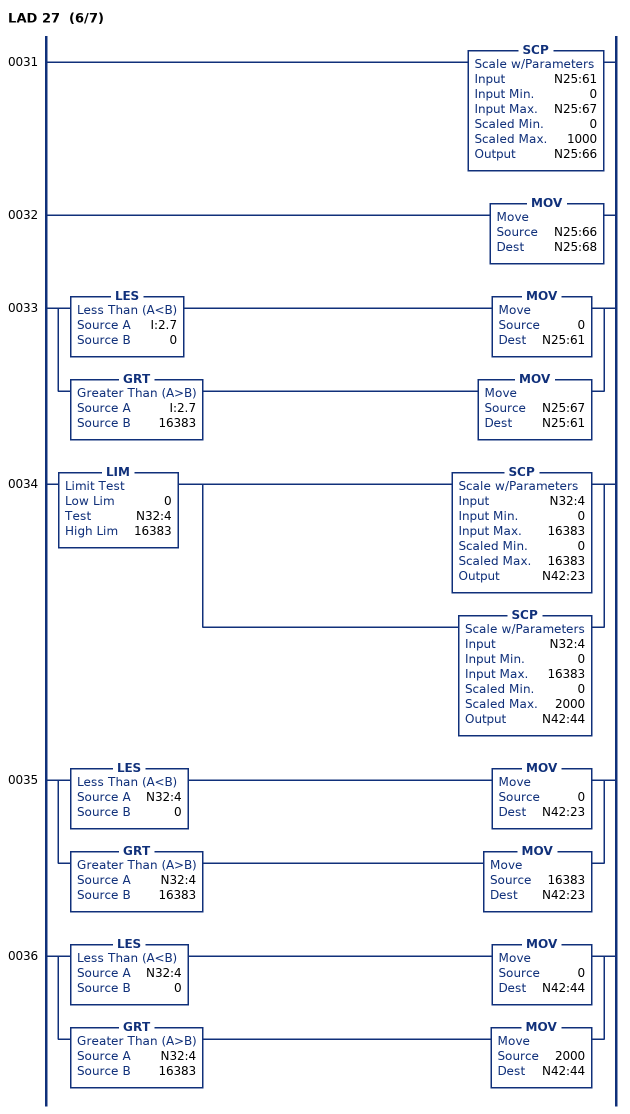
% Rung: 31 %
SOR SCP N25:61 0 N25:67 0 1000 N25:66 EOR
% Rung: 32 %
SOR MOV N25:66 N25:68 EOR
% Rung: 33 %
SOR BST LES I:2.7 0 MOV 0 N25:61 NXB GRT I:2.7 16383 MOV N25:67 N25:61 BND EOR
% Rung: 34 %
SOR LIM 0 N32:4 16383 BST SCP N32:4 0 16383 0 16383 N42:23 NXB SCP N32:4 0 16383 0 2000 N42:44 BND EOR
% Rung: 35 %
SOR BST LES N32:4 0 MOV 0 N42:23 NXB GRT N32:4 16383 MOV 16383 N42:23 BND EOR
% Rung: 36 %
SOR BST LES N32:4 0 MOV 0 N42:44 NXB GRT N32:4 16383 MOV 2000 N42:44 BND EOR

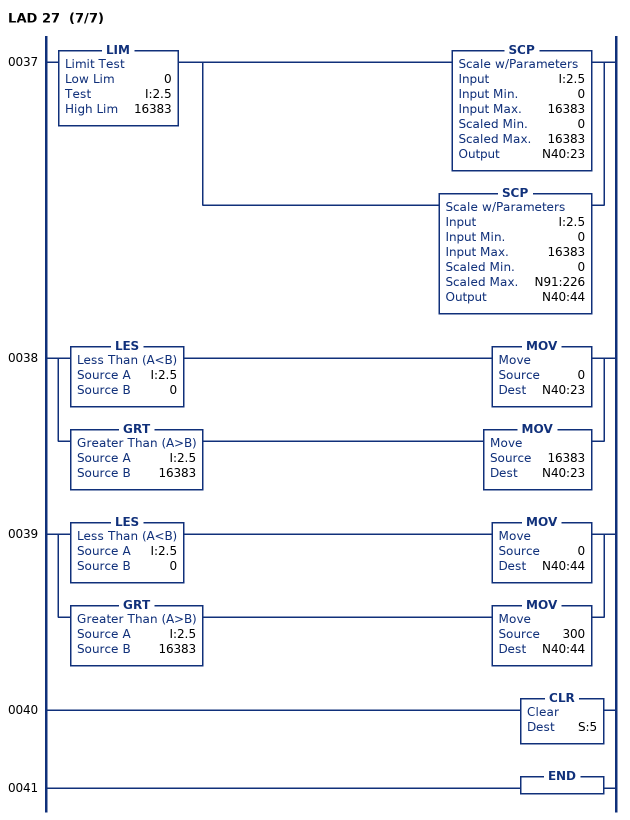
% Rung: 37 %
SOR LIM 0 I:2.5 16383 BST SCP I:2.5 0 16383 0 16383 N40:23 NXB SCP I:2.5 0 16383 0 N91:226 N40:44 BND EOR
% Rung: 38 %
SOR BST LES I:2.5 0 MOV 0 N40:23 NXB GRT I:2.5 16383 MOV 16383 N40:23 BND EOR
% Rung: 39 %
SOR BST LES I:2.5 0 MOV 0 N40:44 NXB GRT I:2.5 16383 MOV 300 N40:44 BND EOR
% Rung: 40 %
SOR CLR S:5 EOR
% Rung: 41 %
SOR END EOR

LADDER 30
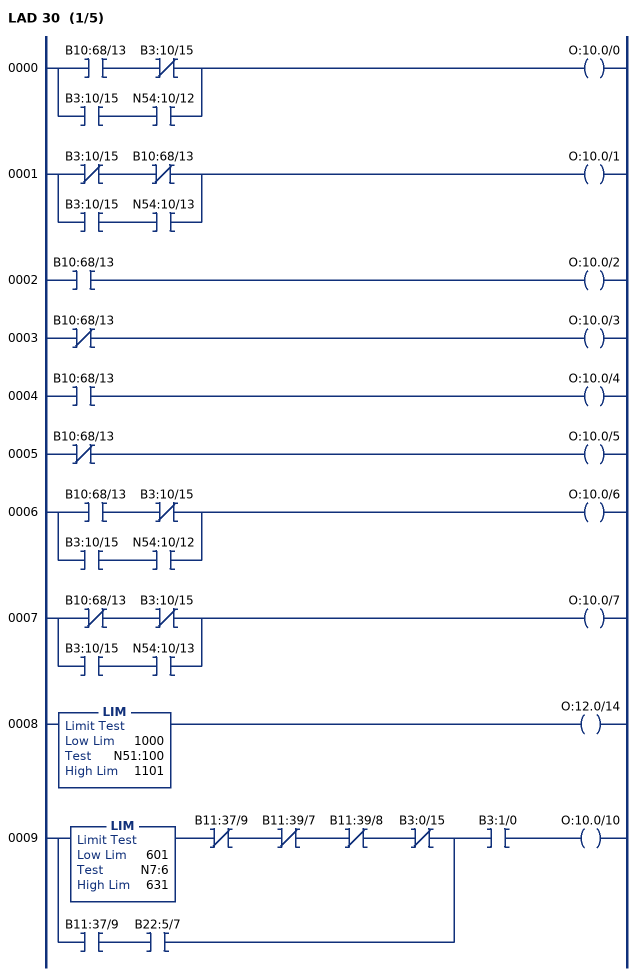
% Rung: 0 %
SOR BST XIC B10:68/13 XIO B3:10/15 NXB XIC B3:10/15 XIC N54:10/12 BND OTE O:10.0/0 EOR
% Rung: 1 %
SOR BST XIO B3:10/15 XIO B10:68/13 NXB XIC B3:10/15 XIC N54:10/13 BND OTE O:10.0/1 EOR
% Rung: 2 %
SOR XIC B10:68/13 OTE O:10.0/2 EOR
% Rung: 3 %
SOR XIO B10:68/13 OTE O:10.0/3 EOR
% Rung: 4 %
SOR XIC B10:68/13 OTE O:10.0/4 EOR
% Rung: 5 %
SOR XIO B10:68/13 OTE O:10.0/5 EOR
% Rung: 6 %
SOR BST XIC B10:68/13 XIO B3:10/15 NXB XIC B3:10/15 XIC N54:10/12 BND OTE O:10.0/6 EOR
% Rung: 7 %
SOR BST XIO B10:68/13 XIO B3:10/15 NXB XIC B3:10/15 XIC N54:10/13 BND OTE O:10.0/7 EOR
% Rung: 8 %
SOR LIM 1000 N51:100 1101 OTE O:12.0/14 EOR
% Rung: 9 %
SOR BST LIM 601 N7:6 631 XIO B11:37/9 XIO B11:39/7 XIO B11:39/8 XIO B3:0/15 NXB XIC B11:37/9 XIC B22:5/7 BND XIC B3:1/0 OTE O:10.0/10 EOR

